% RSLogix 500 project BANCTEST.RSS, saved by version 9.00.00.04 %
PROJECT "BANCTEST"    % processor: SLC 500, 1747-L542 %

PROGRAM FILES
  LAD 2   50 rungs
  LAD 3   16 rungs
  LAD 4   37 rungs
  LAD 5   18 rungs
  LAD 6   36 rungs
  LAD 7   20 rungs
  LAD 8   20 rungs
  LAD 9   15 rungs
  LAD 10   7 rungs
  LAD 11   8 rungs
  LAD 12   10 rungs
  LAD 13   11 rungs
  LAD 14   19 rungs
  LAD 15   13 rungs
  LAD 21   53 rungs
  LAD 22   64 rungs
  LAD 23   50 rungs
  LAD 24   47 rungs
  LAD 16, 17, 18, 19, 20, 25, 26, 27, 28, 29, 30: only END

DATA FILES
  O0 OUTPUT  44 elements
  I1 INPUT  34 elements
  S2 STATUS  164 elements
  B3 BINARY  11 elements
  T4 TIMER  200 elements
  C5 COUNTER  1 elements
  R6 CONTROL  1 elements
  N7 INTEGER  151 elements
  F8 FLOAT  51 elements
  ST20   11 elements
  N21   100 elements
  N22   100 elements
  N23   51 elements
  N31   51 elements
  N32   51 elements
  N33   51 elements
  N34   51 elements
  N35   51 elements
  N36   51 elements
  N37   51 elements
  N38   51 elements
  N39   1 elements
  N40   11 elements
  N41   11 elements
  N50   50 elements
  N51   21 elements

LADDER 2
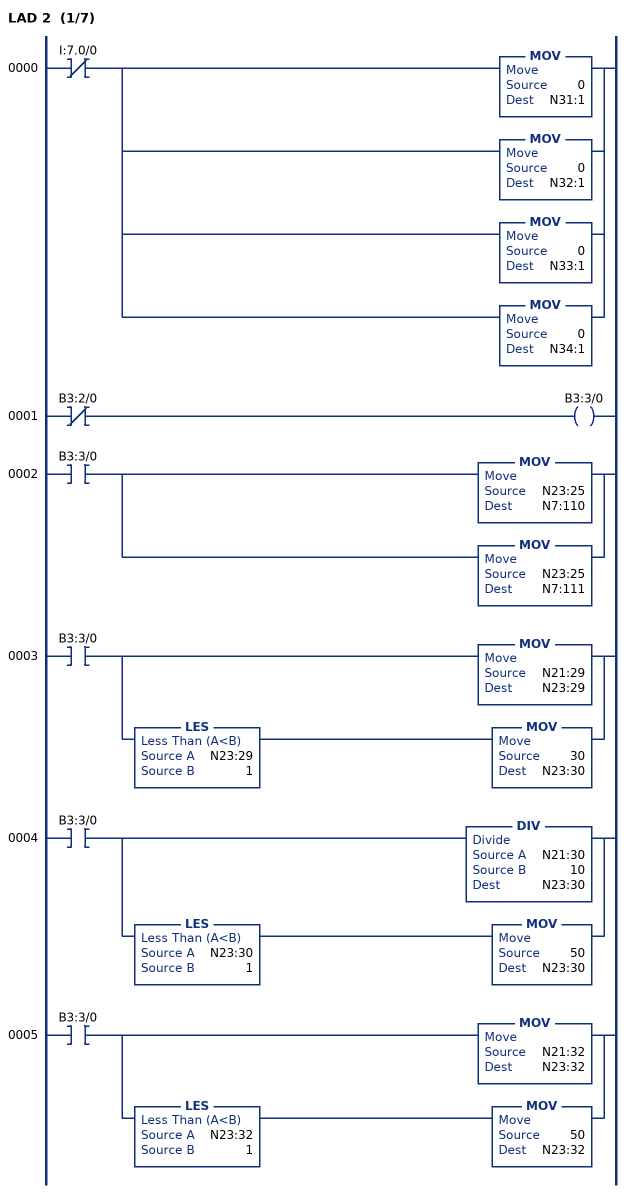
% Rung: 0 %
SOR XIO I:7.0/0 BST MOV 0 N31:1 NXB MOV 0 N32:1 NXB MOV 0 N33:1 NXB MOV 0 N34:1 BND EOR
% Rung: 1 %
SOR XIO B3:2/0 OTE B3:3/0 EOR
% Rung: 2 %
SOR XIC B3:3/0 BST MOV N23:25 N7:110 NXB MOV N23:25 N7:111 BND EOR
% Rung: 3 %
SOR XIC B3:3/0 BST MOV N21:29 N23:29 NXB LES N23:29 1 MOV 30 N23:30 BND EOR
% Rung: 4 %
SOR XIC B3:3/0 BST DIV N21:30 10 N23:30 NXB LES N23:30 1 MOV 50 N23:30 BND EOR
% Rung: 5 %
SOR XIC B3:3/0 BST MOV N21:32 N23:32 NXB LES N23:32 1 MOV 50 N23:32 BND EOR

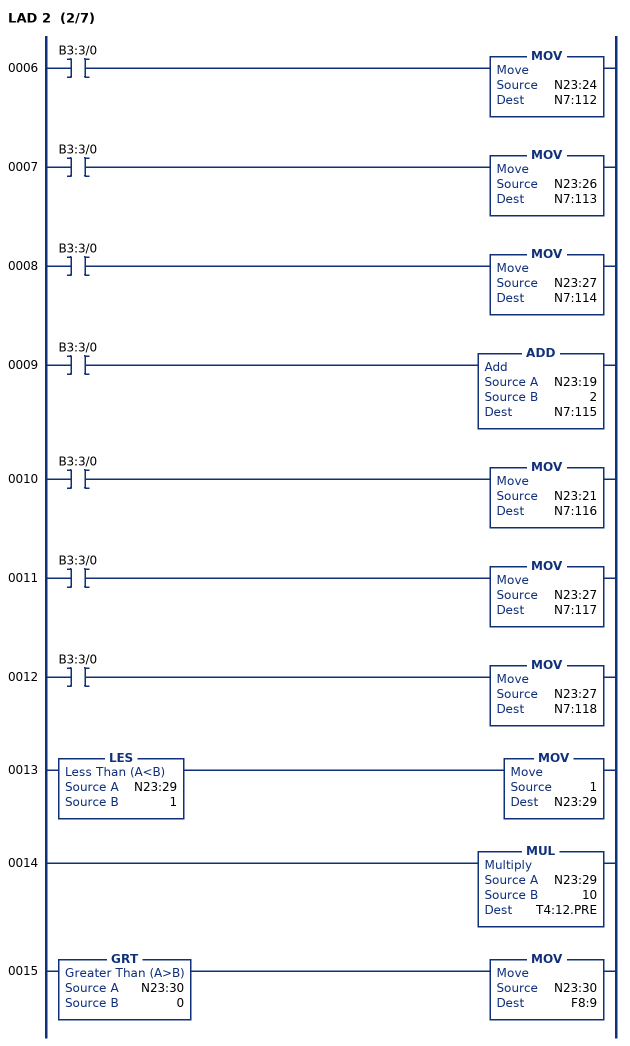
% Rung: 6 %
SOR XIC B3:3/0 MOV N23:24 N7:112 EOR
% Rung: 7 %
SOR XIC B3:3/0 MOV N23:26 N7:113 EOR
% Rung: 8 %
SOR XIC B3:3/0 MOV N23:27 N7:114 EOR
% Rung: 9 %
SOR XIC B3:3/0 ADD N23:19 2 N7:115 EOR
% Rung: 10 %
SOR XIC B3:3/0 MOV N23:21 N7:116 EOR
% Rung: 11 %
SOR XIC B3:3/0 MOV N23:27 N7:117 EOR
% Rung: 12 %
SOR XIC B3:3/0 MOV N23:27 N7:118 EOR
% Rung: 13 %
SOR LES N23:29 1 MOV 1 N23:29 EOR
% Rung: 14 %
SOR MUL N23:29 10 T4:12.PRE EOR
% Rung: 15 %
SOR GRT N23:30 0 MOV N23:30 F8:9 EOR

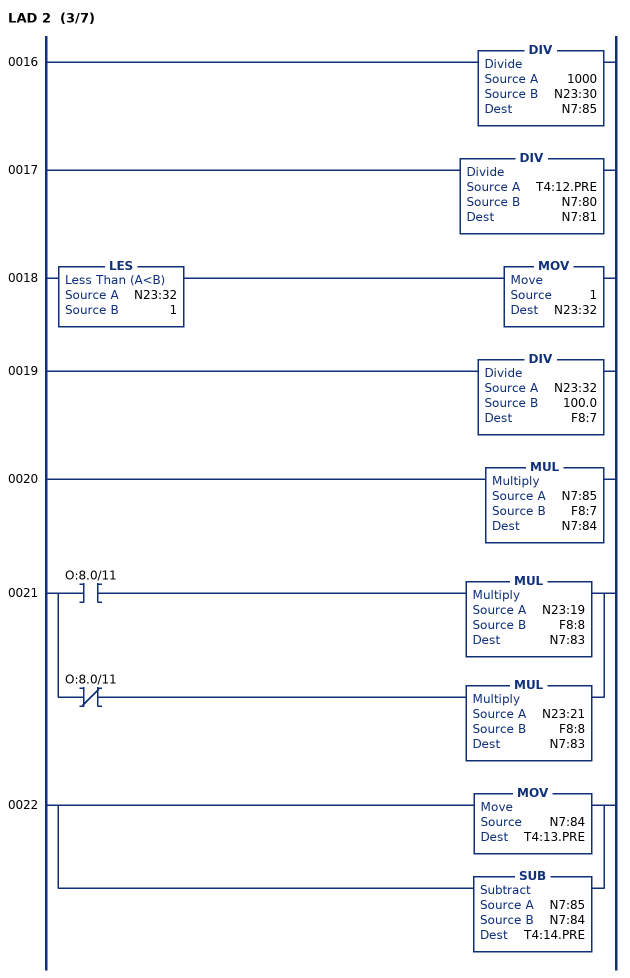
% Rung: 16 %
SOR DIV 1000 N23:30 N7:85 EOR
% Rung: 17 %
SOR DIV T4:12.PRE N7:80 N7:81 EOR
% Rung: 18 %
SOR LES N23:32 1 MOV 1 N23:32 EOR
% Rung: 19 %
SOR DIV N23:32 100.0 F8:7 EOR
% Rung: 20 %
SOR MUL N7:85 F8:7 N7:84 EOR
% Rung: 21 %
SOR BST XIC O:8.0/11 MUL N23:19 F8:8 N7:83 NXB XIO O:8.0/11 MUL N23:21 F8:8 N7:83 BND EOR
% Rung: 22 %
SOR BST MOV N7:84 T4:13.PRE NXB SUB N7:85 N7:84 T4:14.PRE BND EOR

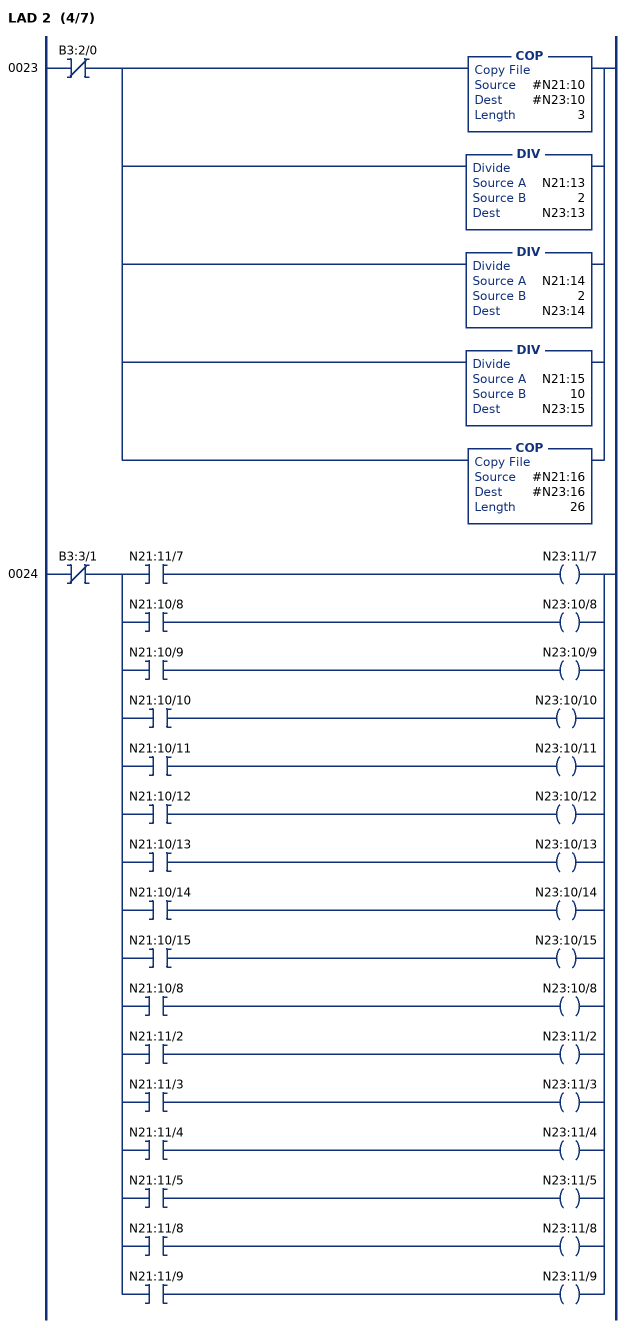
% Rung: 23 %
SOR XIO B3:2/0 BST COP #N21:10 #N23:10 3 NXB DIV N21:13 2 N23:13 NXB DIV N21:14 2 N23:14 NXB DIV N21:15 10 N23:15 NXB COP #N21:16 #N23:16 26 BND EOR
% Rung: 24 %
SOR XIO B3:3/1 BST XIC N21:11/7 OTE N23:11/7 NXB XIC N21:10/8 OTE N23:10/8 NXB XIC N21:10/9 OTE N23:10/9 NXB XIC N21:10/10 OTE N23:10/10 NXB XIC N21:10/11 OTE N23:10/11 NXB XIC N21:10/12 OTE N23:10/12 NXB XIC N21:10/13 OTE N23:10/13 NXB XIC N21:10/14 OTE N23:10/14 NXB XIC N21:10/15 OTE N23:10/15 NXB XIC N21:10/8 OTE N23:10/8 NXB XIC N21:11/2 OTE N23:11/2 NXB XIC N21:11/3 OTE N23:11/3 NXB XIC N21:11/4 OTE N23:11/4 NXB XIC N21:11/5 OTE N23:11/5 NXB XIC N21:11/8 OTE N23:11/8 NXB XIC N21:11/9 OTE N23:11/9 BND EOR

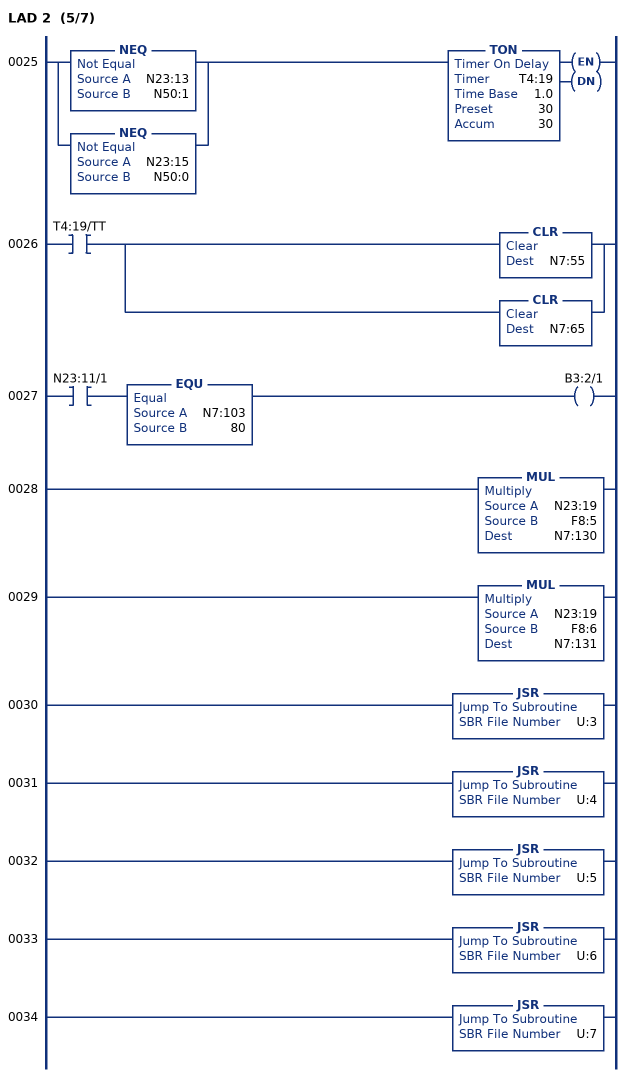
% Rung: 25 %
SOR BST NEQ N23:13 N50:1 NXB NEQ N23:15 N50:0 BND TON T4:19 1.0 30 30 EOR
% Rung: 26 %
SOR XIC T4:19/TT BST CLR N7:55 NXB CLR N7:65 BND EOR
% Rung: 27 %
SOR XIC N23:11/1 EQU N7:103 80 OTE B3:2/1 EOR
% Rung: 28 %
SOR MUL N23:19 F8:5 N7:130 EOR
% Rung: 29 %
SOR MUL N23:19 F8:6 N7:131 EOR
% Rung: 30 %
SOR JSR U:3 EOR
% Rung: 31 %
SOR JSR U:4 EOR
% Rung: 32 %
SOR JSR U:5 EOR
% Rung: 33 %
SOR JSR U:6 EOR
% Rung: 34 %
SOR JSR U:7 EOR

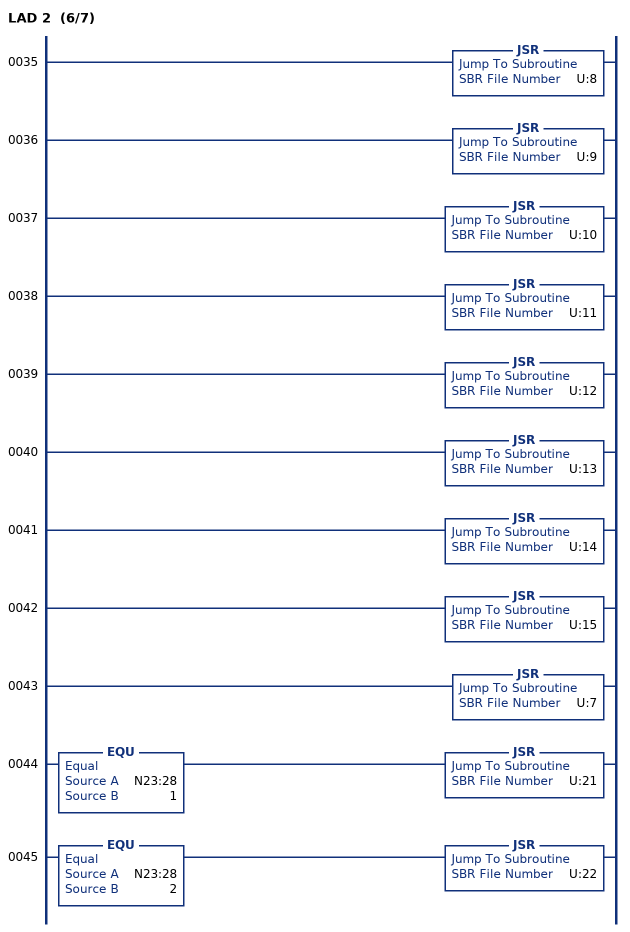
% Rung: 35 %
SOR JSR U:8 EOR
% Rung: 36 %
SOR JSR U:9 EOR
% Rung: 37 %
SOR JSR U:10 EOR
% Rung: 38 %
SOR JSR U:11 EOR
% Rung: 39 %
SOR JSR U:12 EOR
% Rung: 40 %
SOR JSR U:13 EOR
% Rung: 41 %
SOR JSR U:14 EOR
% Rung: 42 %
SOR JSR U:15 EOR
% Rung: 43 %
SOR JSR U:7 EOR
% Rung: 44 %
SOR EQU N23:28 1 JSR U:21 EOR
% Rung: 45 %
SOR EQU N23:28 2 JSR U:22 EOR

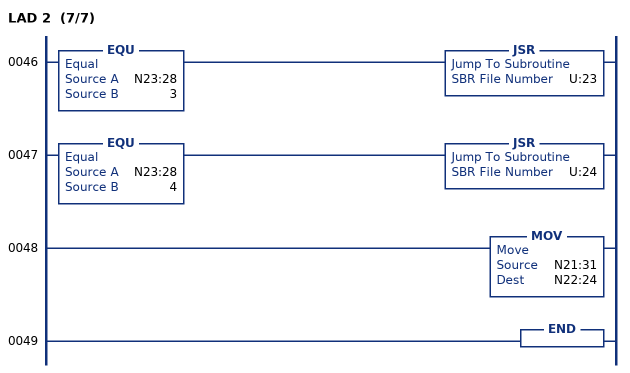
% Rung: 46 %
SOR EQU N23:28 3 JSR U:23 EOR
% Rung: 47 %
SOR EQU N23:28 4 JSR U:24 EOR
% Rung: 48 %
SOR MOV N21:31 N22:24 EOR
% Rung: 49 %
SOR END EOR

LADDER 3
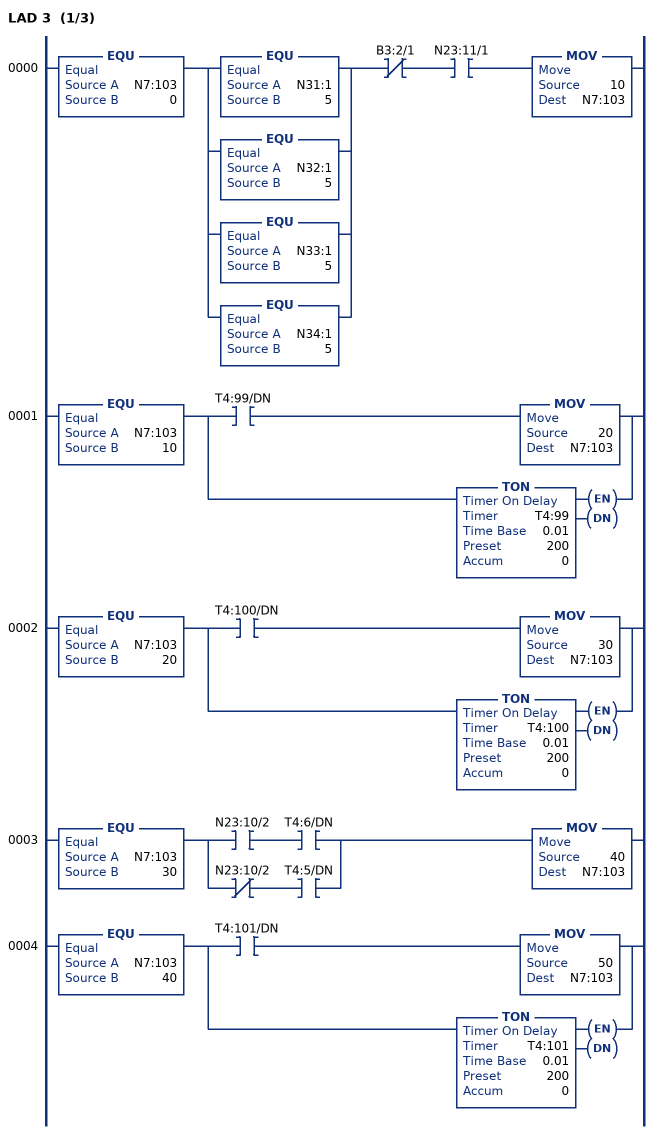
% Rung: 0 %
SOR EQU N7:103 0 BST EQU N31:1 5 NXB EQU N32:1 5 NXB EQU N33:1 5 NXB EQU N34:1 5 BND XIO B3:2/1 XIC N23:11/1 MOV 10 N7:103 EOR
% Rung: 1 %
SOR EQU N7:103 10 BST XIC T4:99/DN MOV 20 N7:103 NXB TON T4:99 0.01 200 0 BND EOR
% Rung: 2 %
SOR EQU N7:103 20 BST XIC T4:100/DN MOV 30 N7:103 NXB TON T4:100 0.01 200 0 BND EOR
% Rung: 3 %
SOR EQU N7:103 30 BST XIC N23:10/2 XIC T4:6/DN NXB XIO N23:10/2 XIC T4:5/DN BND MOV 40 N7:103 EOR
% Rung: 4 %
SOR EQU N7:103 40 BST XIC T4:101/DN MOV 50 N7:103 NXB TON T4:101 0.01 200 0 BND EOR

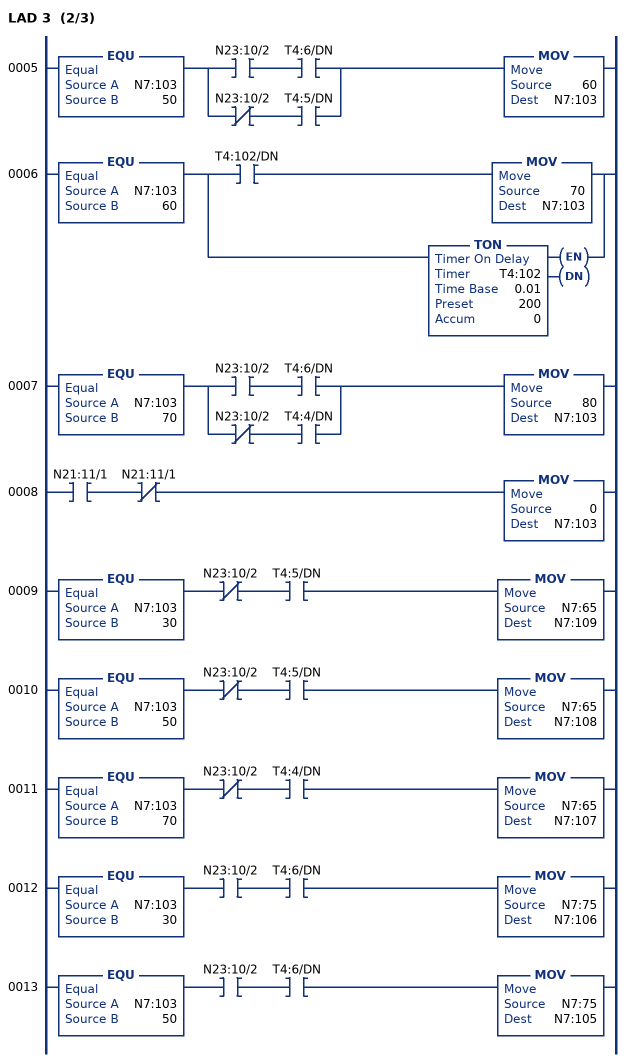
% Rung: 5 %
SOR EQU N7:103 50 BST XIC N23:10/2 XIC T4:6/DN NXB XIO N23:10/2 XIC T4:5/DN BND MOV 60 N7:103 EOR
% Rung: 6 %
SOR EQU N7:103 60 BST XIC T4:102/DN MOV 70 N7:103 NXB TON T4:102 0.01 200 0 BND EOR
% Rung: 7 %
SOR EQU N7:103 70 BST XIC N23:10/2 XIC T4:6/DN NXB XIO N23:10/2 XIC T4:4/DN BND MOV 80 N7:103 EOR
% Rung: 8 %
SOR XIC N21:11/1 XIO N21:11/1 MOV 0 N7:103 EOR
% Rung: 9 %
SOR EQU N7:103 30 XIO N23:10/2 XIC T4:5/DN MOV N7:65 N7:109 EOR
% Rung: 10 %
SOR EQU N7:103 50 XIO N23:10/2 XIC T4:5/DN MOV N7:65 N7:108 EOR
% Rung: 11 %
SOR EQU N7:103 70 XIO N23:10/2 XIC T4:4/DN MOV N7:65 N7:107 EOR
% Rung: 12 %
SOR EQU N7:103 30 XIC N23:10/2 XIC T4:6/DN MOV N7:75 N7:106 EOR
% Rung: 13 %
SOR EQU N7:103 50 XIC N23:10/2 XIC T4:6/DN MOV N7:75 N7:105 EOR

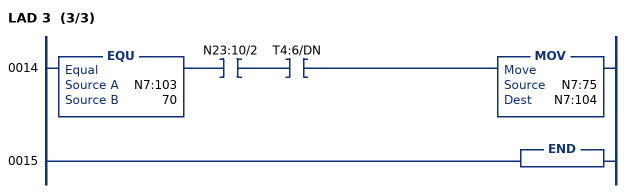
% Rung: 14 %
SOR EQU N7:103 70 XIC N23:10/2 XIC T4:6/DN MOV N7:75 N7:104 EOR
% Rung: 15 %
SOR END EOR

LADDER 4
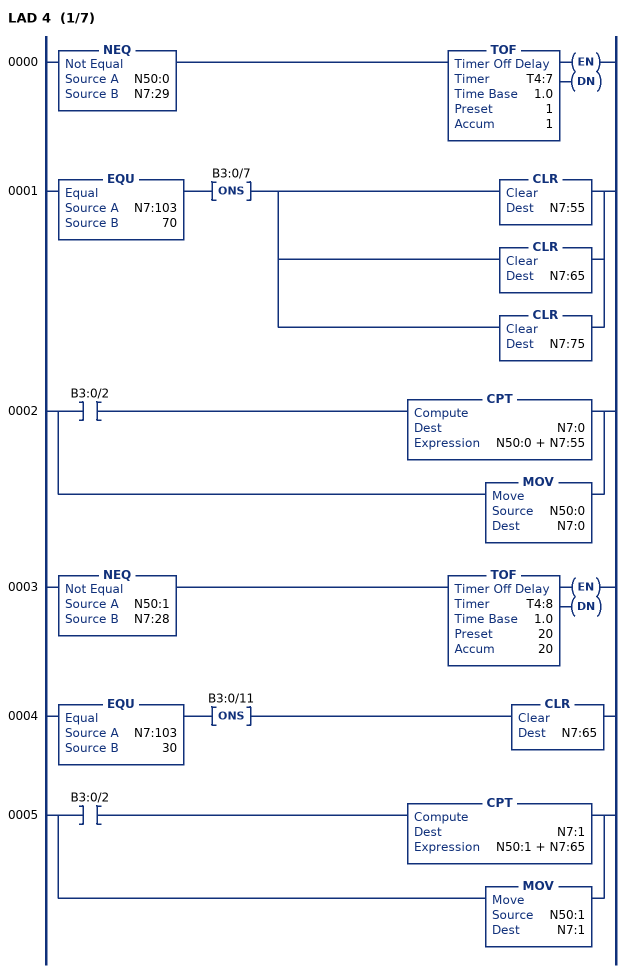
% Rung: 0 %
SOR NEQ N50:0 N7:29 TOF T4:7 1.0 1 1 EOR
% Rung: 1 %
SOR EQU N7:103 70 OSR B3:0/7 BST CLR N7:55 NXB CLR N7:65 NXB CLR N7:75 BND EOR
% Rung: 2 %
SOR BST XIC B3:0/2 CPT N7:0 " N50:0 + N7:55 " NXB MOV N50:0 N7:0 BND EOR
% Rung: 3 %
SOR NEQ N50:1 N7:28 TOF T4:8 1.0 20 20 EOR
% Rung: 4 %
SOR EQU N7:103 30 OSR B3:0/11 CLR N7:65 EOR
% Rung: 5 %
SOR BST XIC B3:0/2 CPT N7:1 " N50:1 + N7:65 " NXB MOV N50:1 N7:1 BND EOR

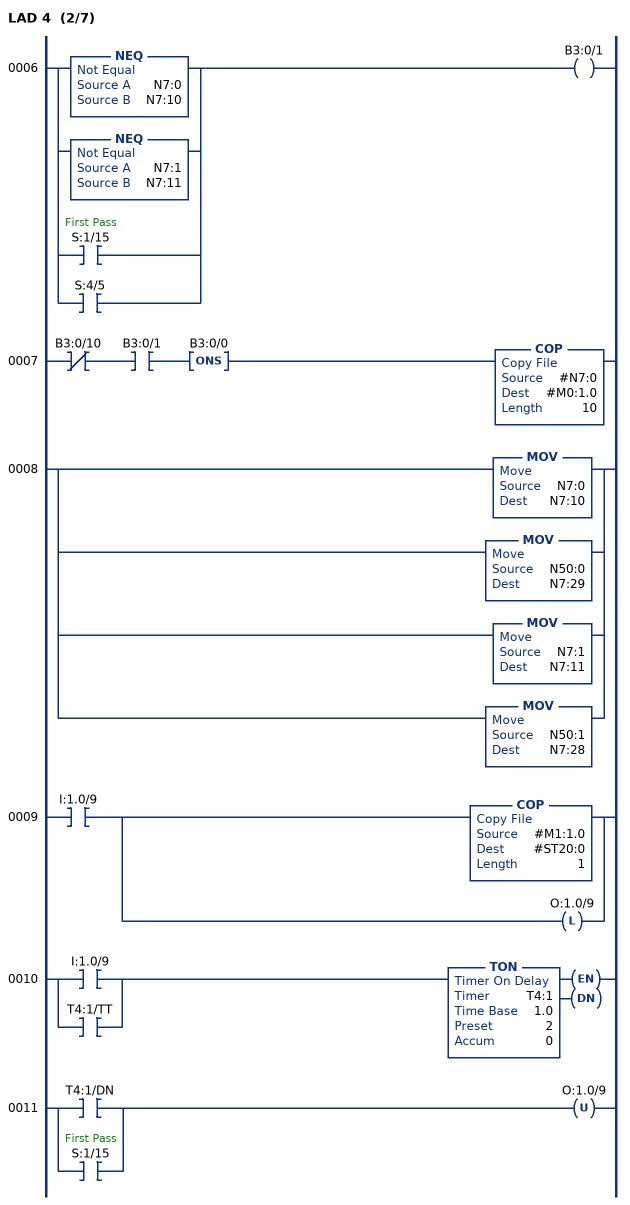
% Rung: 6 %
SOR BST NEQ N7:0 N7:10 NXB NEQ N7:1 N7:11 NXB XIC S:1/15 NXB XIC S:4/5 BND OTE B3:0/1 EOR
%   S:1/15  "First Pass" %
% Rung: 7 %
SOR XIO B3:0/10 XIC B3:0/1 OSR B3:0/0 COP #N7:0 #M0:1.0 10 EOR
% Rung: 8 %
SOR BST MOV N7:0 N7:10 NXB MOV N50:0 N7:29 NXB MOV N7:1 N7:11 NXB MOV N50:1 N7:28 BND EOR
% Rung: 9 %
SOR XIC I:1.0/9 BST COP #M1:1.0 #ST20:0 1 NXB OTL O:1.0/9 BND EOR
% Rung: 10 %
SOR BST XIC I:1.0/9 NXB XIC T4:1/TT BND TON T4:1 1.0 2 0 EOR
% Rung: 11 %
SOR BST XIC T4:1/DN NXB XIC S:1/15 BND OTU O:1.0/9 EOR
%   S:1/15  "First Pass" %

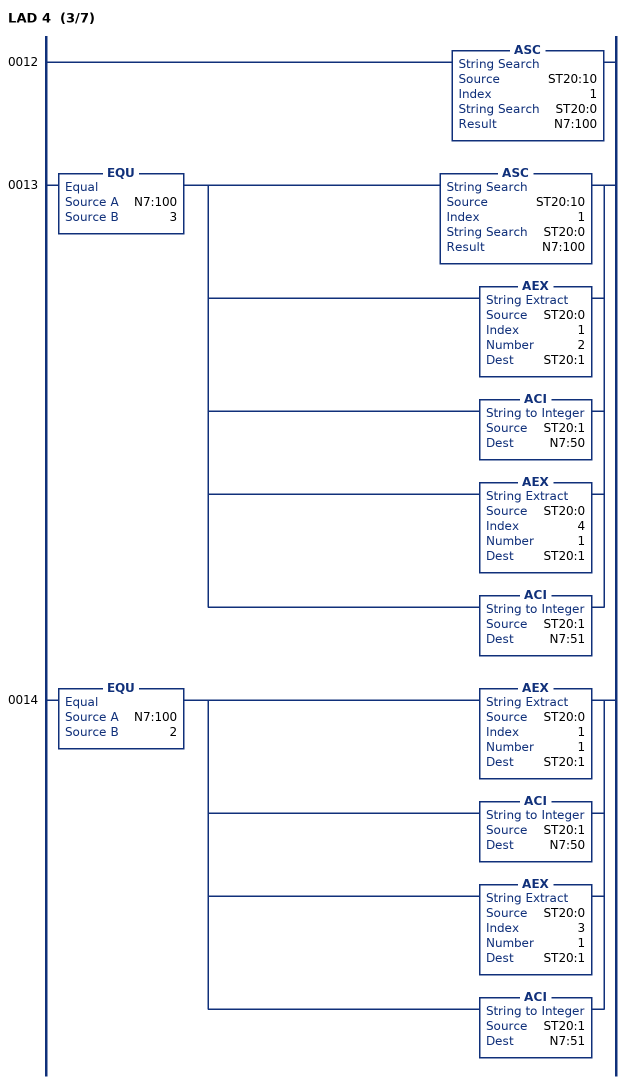
% Rung: 12 %
SOR ASC ST20:10 1 ST20:0 N7:100 EOR
% Rung: 13 %
SOR EQU N7:100 3 BST ASC ST20:10 1 ST20:0 N7:100 NXB AEX ST20:0 1 2 ST20:1 NXB ACI ST20:1 N7:50 NXB AEX ST20:0 4 1 ST20:1 NXB ACI ST20:1 N7:51 BND EOR
% Rung: 14 %
SOR EQU N7:100 2 BST AEX ST20:0 1 1 ST20:1 NXB ACI ST20:1 N7:50 NXB AEX ST20:0 3 1 ST20:1 NXB ACI ST20:1 N7:51 BND EOR

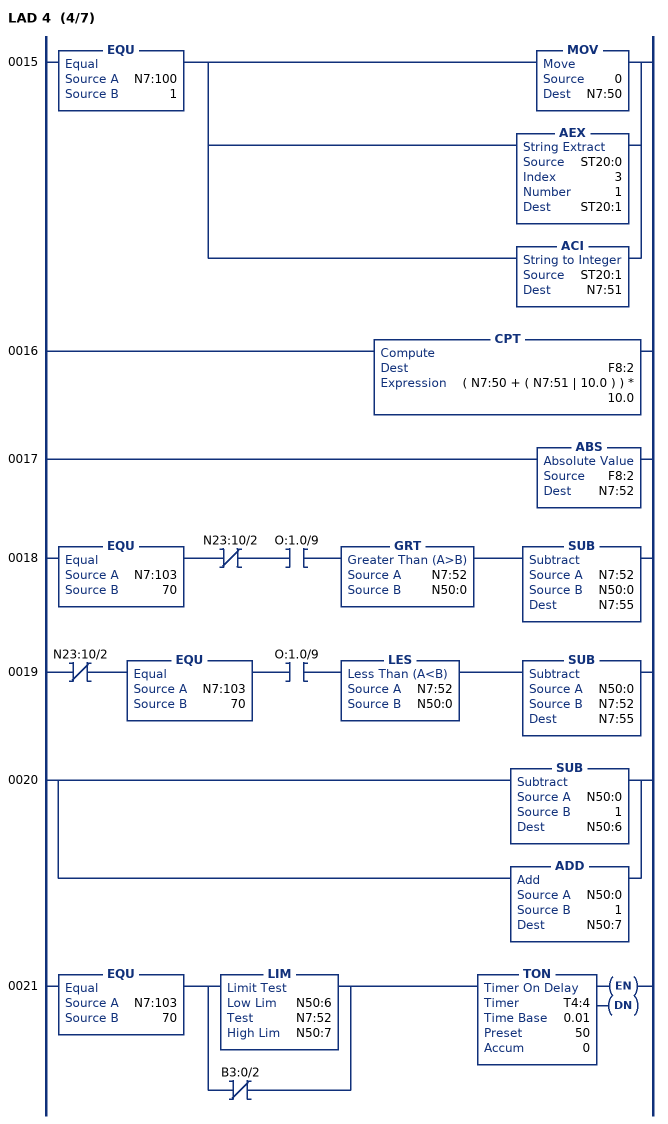
% Rung: 15 %
SOR EQU N7:100 1 BST MOV 0 N7:50 NXB AEX ST20:0 3 1 ST20:1 NXB ACI ST20:1 N7:51 BND EOR
% Rung: 16 %
SOR CPT F8:2 " ( N7:50 + ( N7:51 | 10.0 ) ) * 10.0 " EOR
% Rung: 17 %
SOR ABS F8:2 N7:52 EOR
% Rung: 18 %
SOR EQU N7:103 70 XIO N23:10/2 XIC O:1.0/9 GRT N7:52 N50:0 SUB N7:52 N50:0 N7:55 EOR
% Rung: 19 %
SOR XIO N23:10/2 EQU N7:103 70 XIC O:1.0/9 LES N7:52 N50:0 SUB N50:0 N7:52 N7:55 EOR
% Rung: 20 %
SOR BST SUB N50:0 1 N50:6 NXB ADD N50:0 1 N50:7 BND EOR
% Rung: 21 %
SOR EQU N7:103 70 BST LIM N50:6 N7:52 N50:7 NXB XIO B3:0/2 BND TON T4:4 0.01 50 0 EOR

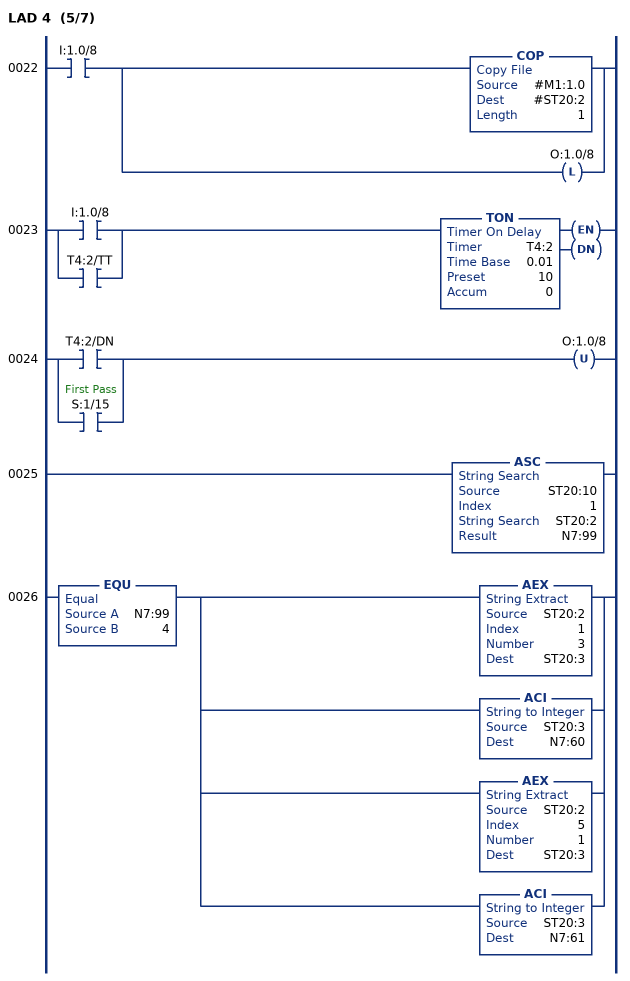
% Rung: 22 %
SOR XIC I:1.0/8 BST COP #M1:1.0 #ST20:2 1 NXB OTL O:1.0/8 BND EOR
% Rung: 23 %
SOR BST XIC I:1.0/8 NXB XIC T4:2/TT BND TON T4:2 0.01 10 0 EOR
% Rung: 24 %
SOR BST XIC T4:2/DN NXB XIC S:1/15 BND OTU O:1.0/8 EOR
%   S:1/15  "First Pass" %
% Rung: 25 %
SOR ASC ST20:10 1 ST20:2 N7:99 EOR
% Rung: 26 %
SOR EQU N7:99 4 BST AEX ST20:2 1 3 ST20:3 NXB ACI ST20:3 N7:60 NXB AEX ST20:2 5 1 ST20:3 NXB ACI ST20:3 N7:61 BND EOR

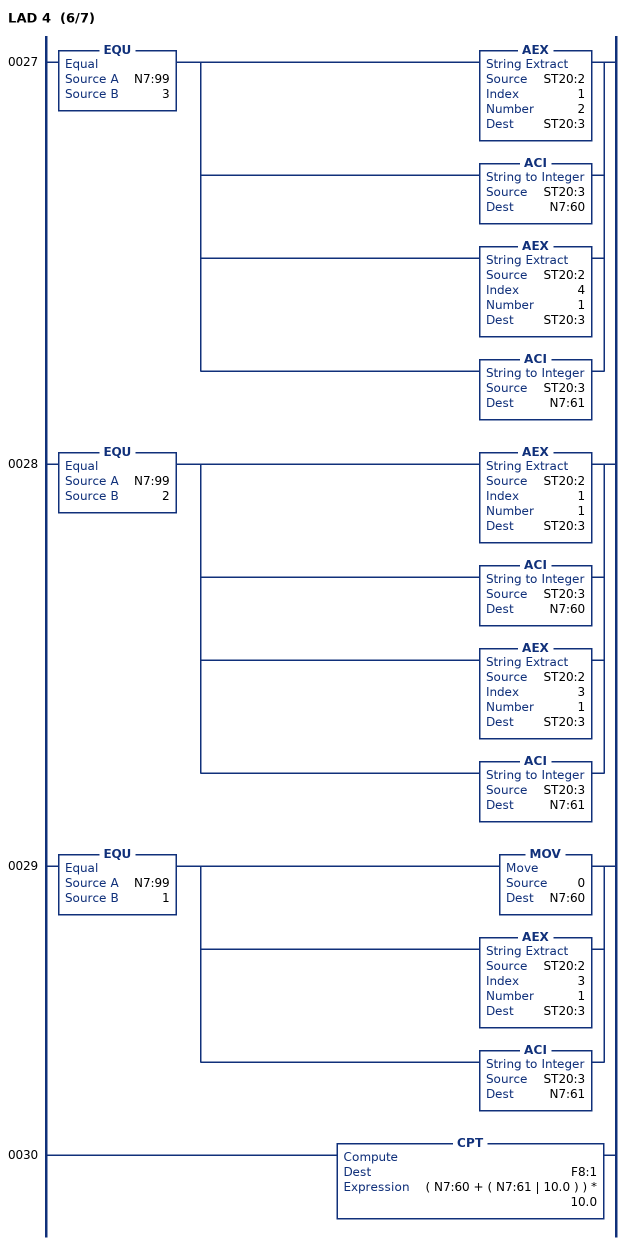
% Rung: 27 %
SOR EQU N7:99 3 BST AEX ST20:2 1 2 ST20:3 NXB ACI ST20:3 N7:60 NXB AEX ST20:2 4 1 ST20:3 NXB ACI ST20:3 N7:61 BND EOR
% Rung: 28 %
SOR EQU N7:99 2 BST AEX ST20:2 1 1 ST20:3 NXB ACI ST20:3 N7:60 NXB AEX ST20:2 3 1 ST20:3 NXB ACI ST20:3 N7:61 BND EOR
% Rung: 29 %
SOR EQU N7:99 1 BST MOV 0 N7:60 NXB AEX ST20:2 3 1 ST20:3 NXB ACI ST20:3 N7:61 BND EOR
% Rung: 30 %
SOR CPT F8:1 " ( N7:60 + ( N7:61 | 10.0 ) ) * 10.0 " EOR

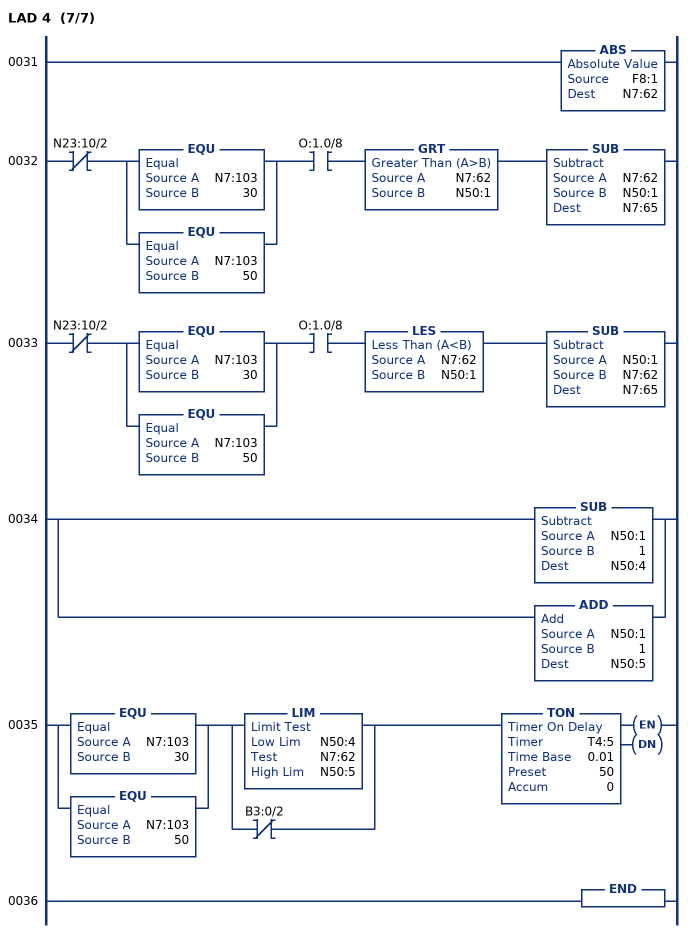
% Rung: 31 %
SOR ABS F8:1 N7:62 EOR
% Rung: 32 %
SOR XIO N23:10/2 BST EQU N7:103 30 NXB EQU N7:103 50 BND XIC O:1.0/8 GRT N7:62 N50:1 SUB N7:62 N50:1 N7:65 EOR
% Rung: 33 %
SOR XIO N23:10/2 BST EQU N7:103 30 NXB EQU N7:103 50 BND XIC O:1.0/8 LES N7:62 N50:1 SUB N50:1 N7:62 N7:65 EOR
% Rung: 34 %
SOR BST SUB N50:1 1 N50:4 NXB ADD N50:1 1 N50:5 BND EOR
% Rung: 35 %
SOR BST EQU N7:103 30 NXB EQU N7:103 50 BND BST LIM N50:4 N7:62 N50:5 NXB XIO B3:0/2 BND TON T4:5 0.01 50 0 EOR
% Rung: 36 %
SOR END EOR

LADDER 5
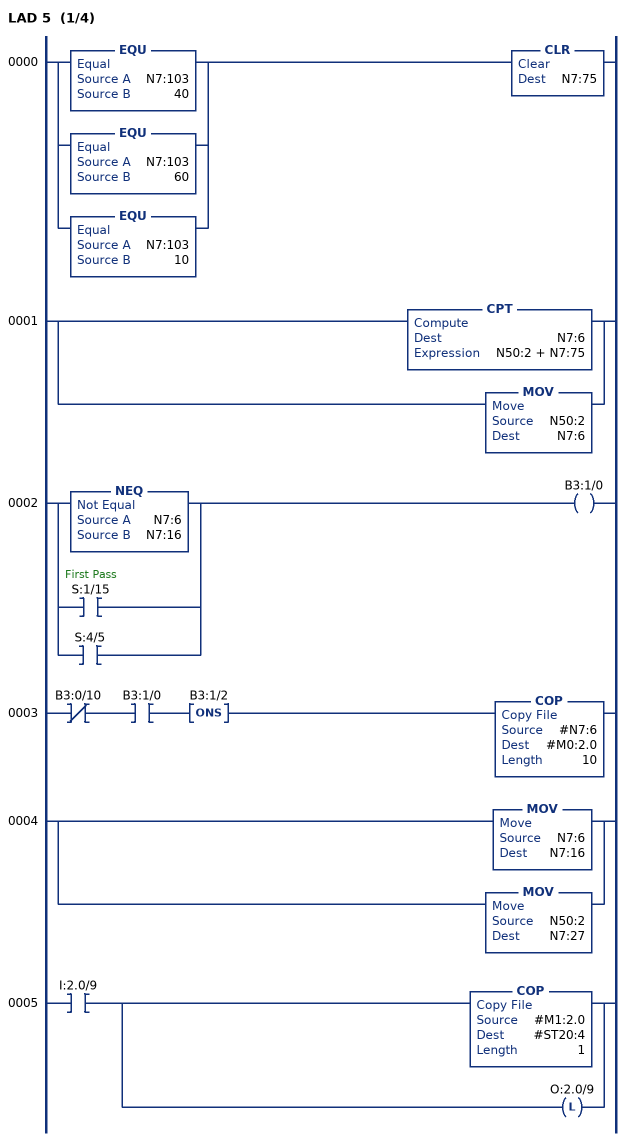
% Rung: 0 %
SOR BST EQU N7:103 40 NXB EQU N7:103 60 NXB EQU N7:103 10 BND CLR N7:75 EOR
% Rung: 1 %
SOR BST CPT N7:6 " N50:2 + N7:75 " NXB MOV N50:2 N7:6 BND EOR
% Rung: 2 %
SOR BST NEQ N7:6 N7:16 NXB XIC S:1/15 NXB XIC S:4/5 BND OTE B3:1/0 EOR
%   S:1/15  "First Pass" %
% Rung: 3 %
SOR XIO B3:0/10 XIC B3:1/0 OSR B3:1/2 COP #N7:6 #M0:2.0 10 EOR
% Rung: 4 %
SOR BST MOV N7:6 N7:16 NXB MOV N50:2 N7:27 BND EOR
% Rung: 5 %
SOR XIC I:2.0/9 BST COP #M1:2.0 #ST20:4 1 NXB OTL O:2.0/9 BND EOR

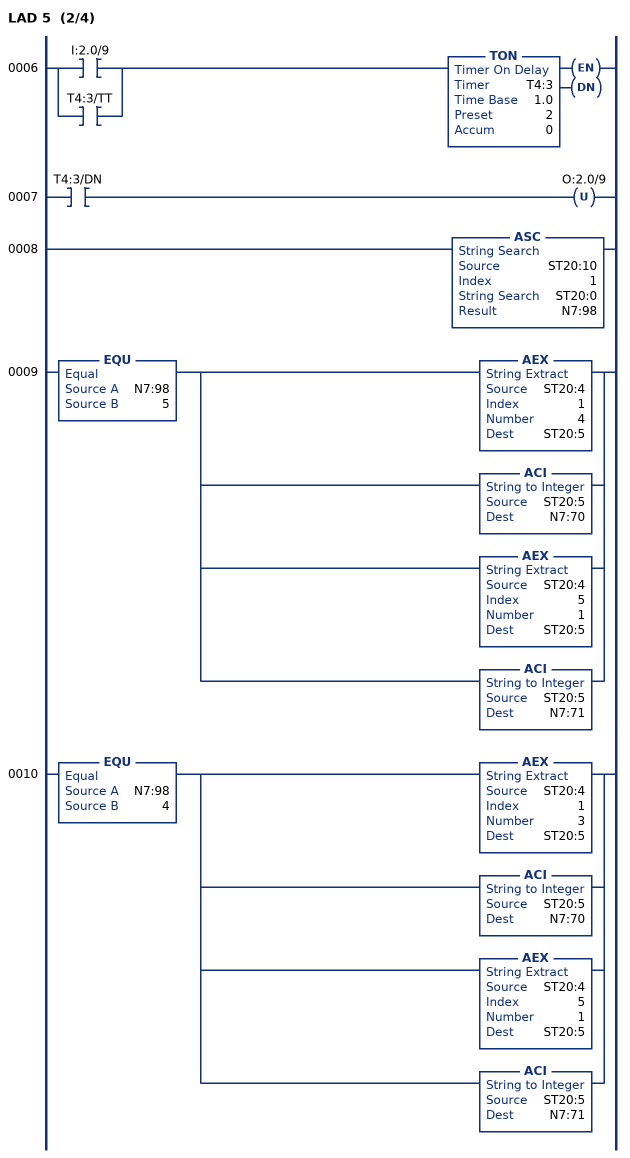
% Rung: 6 %
SOR BST XIC I:2.0/9 NXB XIC T4:3/TT BND TON T4:3 1.0 2 0 EOR
% Rung: 7 %
SOR XIC T4:3/DN OTU O:2.0/9 EOR
% Rung: 8 %
SOR ASC ST20:10 1 ST20:0 N7:98 EOR
% Rung: 9 %
SOR EQU N7:98 5 BST AEX ST20:4 1 4 ST20:5 NXB ACI ST20:5 N7:70 NXB AEX ST20:4 5 1 ST20:5 NXB ACI ST20:5 N7:71 BND EOR
% Rung: 10 %
SOR EQU N7:98 4 BST AEX ST20:4 1 3 ST20:5 NXB ACI ST20:5 N7:70 NXB AEX ST20:4 5 1 ST20:5 NXB ACI ST20:5 N7:71 BND EOR

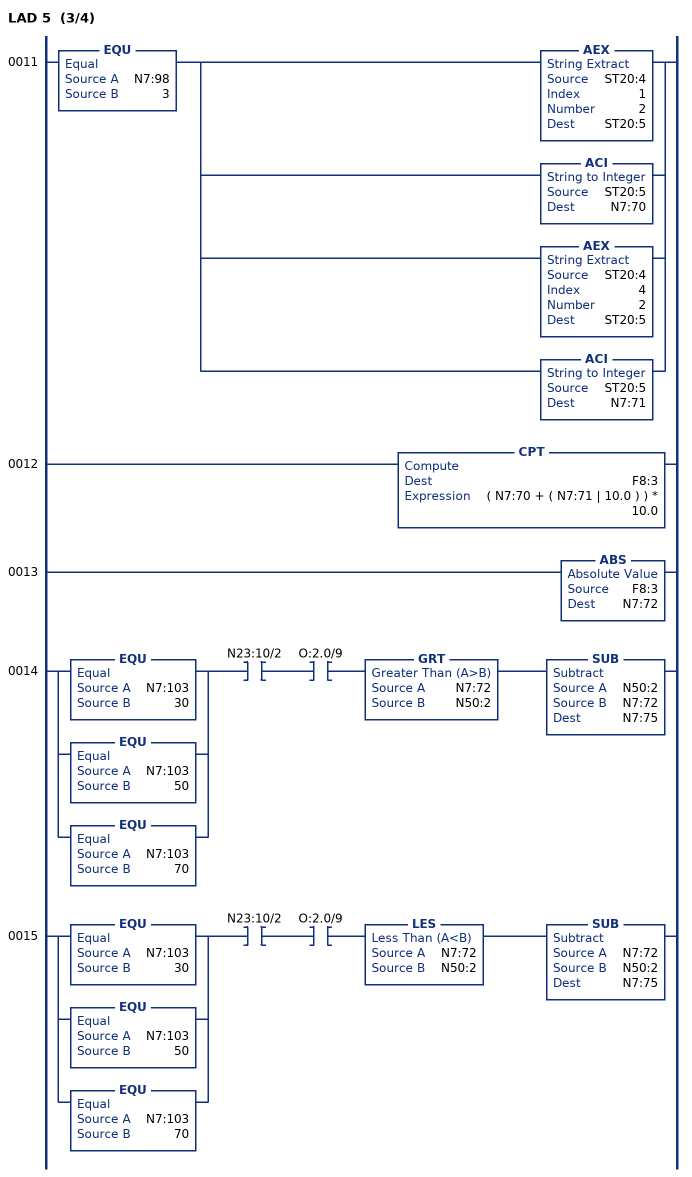
% Rung: 11 %
SOR EQU N7:98 3 BST AEX ST20:4 1 2 ST20:5 NXB ACI ST20:5 N7:70 NXB AEX ST20:4 4 2 ST20:5 NXB ACI ST20:5 N7:71 BND EOR
% Rung: 12 %
SOR CPT F8:3 " ( N7:70 + ( N7:71 | 10.0 ) ) * 10.0 " EOR
% Rung: 13 %
SOR ABS F8:3 N7:72 EOR
% Rung: 14 %
SOR BST EQU N7:103 30 NXB EQU N7:103 50 NXB EQU N7:103 70 BND XIC N23:10/2 XIC O:2.0/9 GRT N7:72 N50:2 SUB N50:2 N7:72 N7:75 EOR
% Rung: 15 %
SOR BST EQU N7:103 30 NXB EQU N7:103 50 NXB EQU N7:103 70 BND XIC N23:10/2 XIC O:2.0/9 LES N7:72 N50:2 SUB N7:72 N50:2 N7:75 EOR

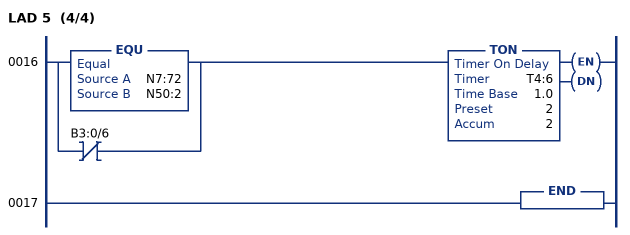
% Rung: 16 %
SOR BST EQU N7:72 N50:2 NXB XIO B3:0/6 BND TON T4:6 1.0 2 2 EOR
% Rung: 17 %
SOR END EOR

LADDER 6
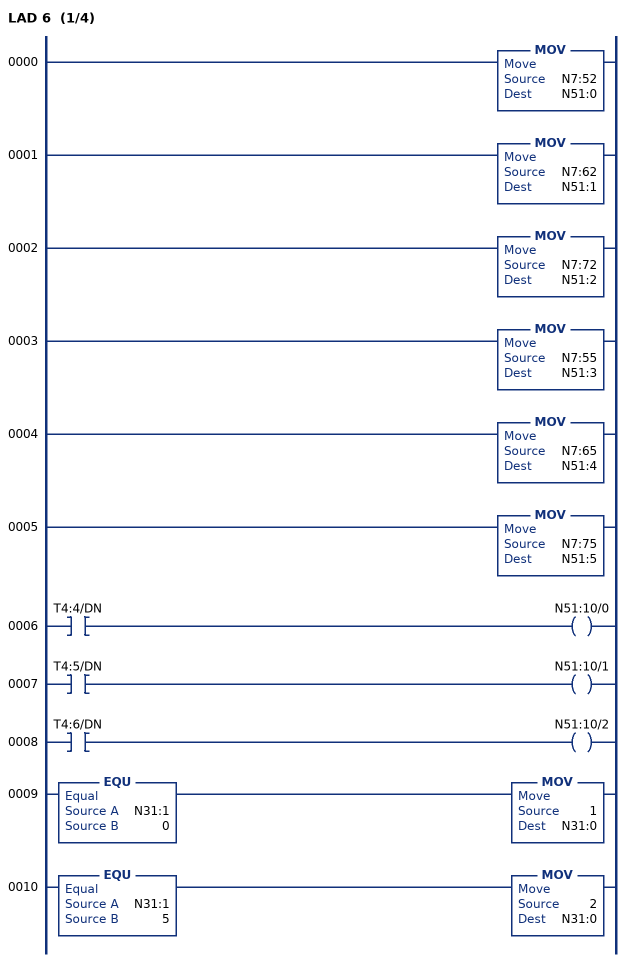
% Rung: 0 %
SOR MOV N7:52 N51:0 EOR
% Rung: 1 %
SOR MOV N7:62 N51:1 EOR
% Rung: 2 %
SOR MOV N7:72 N51:2 EOR
% Rung: 3 %
SOR MOV N7:55 N51:3 EOR
% Rung: 4 %
SOR MOV N7:65 N51:4 EOR
% Rung: 5 %
SOR MOV N7:75 N51:5 EOR
% Rung: 6 %
SOR XIC T4:4/DN OTE N51:10/0 EOR
% Rung: 7 %
SOR XIC T4:5/DN OTE N51:10/1 EOR
% Rung: 8 %
SOR XIC T4:6/DN OTE N51:10/2 EOR
% Rung: 9 %
SOR EQU N31:1 0 MOV 1 N31:0 EOR
% Rung: 10 %
SOR EQU N31:1 5 MOV 2 N31:0 EOR

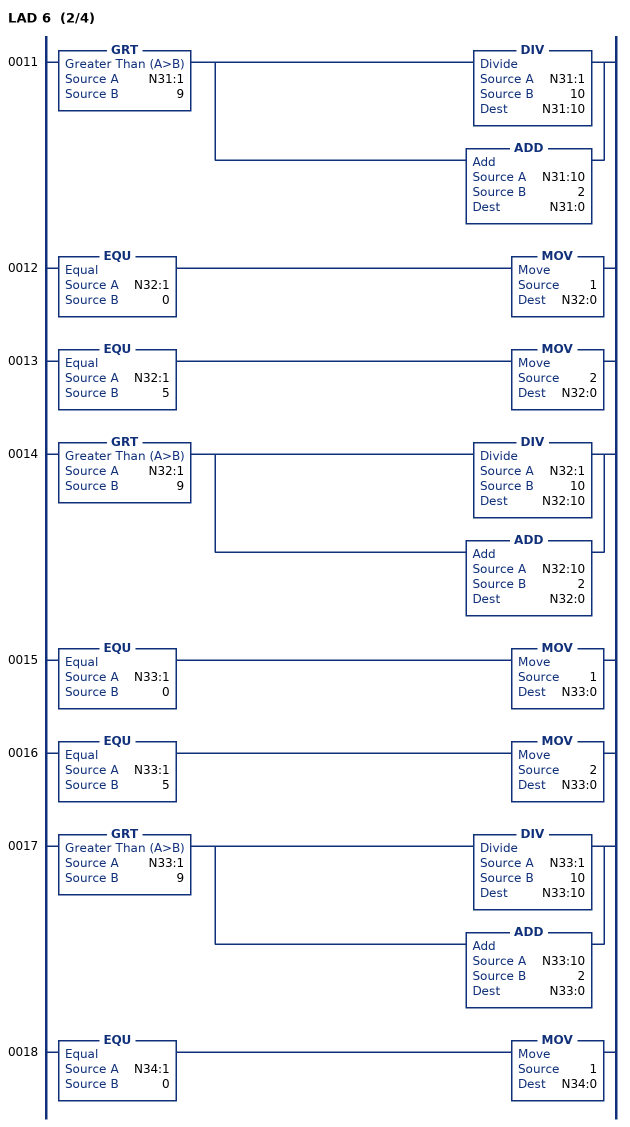
% Rung: 11 %
SOR GRT N31:1 9 BST DIV N31:1 10 N31:10 NXB ADD N31:10 2 N31:0 BND EOR
% Rung: 12 %
SOR EQU N32:1 0 MOV 1 N32:0 EOR
% Rung: 13 %
SOR EQU N32:1 5 MOV 2 N32:0 EOR
% Rung: 14 %
SOR GRT N32:1 9 BST DIV N32:1 10 N32:10 NXB ADD N32:10 2 N32:0 BND EOR
% Rung: 15 %
SOR EQU N33:1 0 MOV 1 N33:0 EOR
% Rung: 16 %
SOR EQU N33:1 5 MOV 2 N33:0 EOR
% Rung: 17 %
SOR GRT N33:1 9 BST DIV N33:1 10 N33:10 NXB ADD N33:10 2 N33:0 BND EOR
% Rung: 18 %
SOR EQU N34:1 0 MOV 1 N34:0 EOR

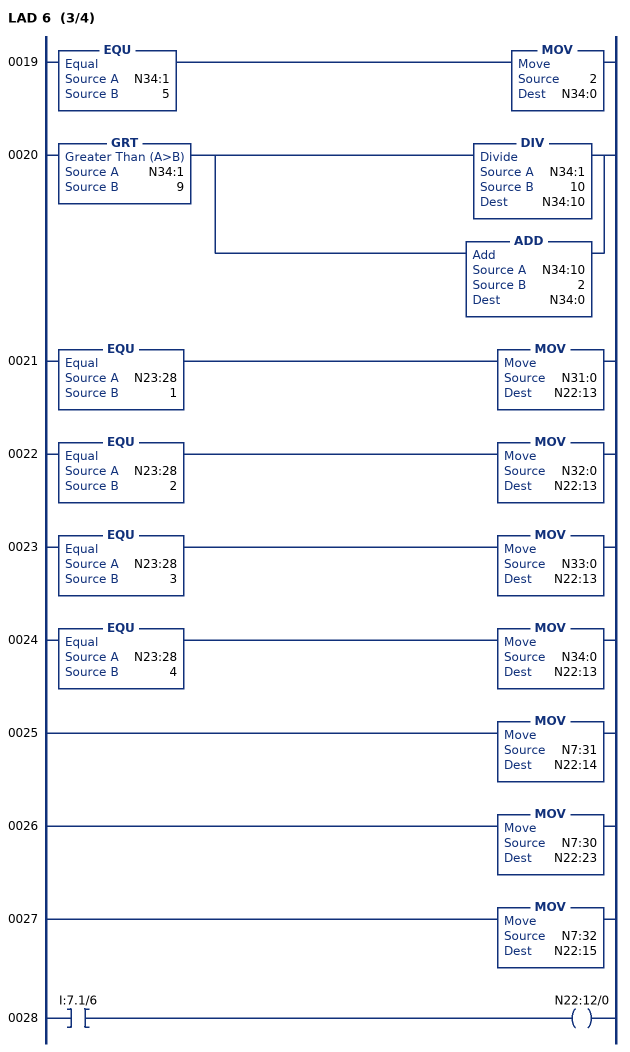
% Rung: 19 %
SOR EQU N34:1 5 MOV 2 N34:0 EOR
% Rung: 20 %
SOR GRT N34:1 9 BST DIV N34:1 10 N34:10 NXB ADD N34:10 2 N34:0 BND EOR
% Rung: 21 %
SOR EQU N23:28 1 MOV N31:0 N22:13 EOR
% Rung: 22 %
SOR EQU N23:28 2 MOV N32:0 N22:13 EOR
% Rung: 23 %
SOR EQU N23:28 3 MOV N33:0 N22:13 EOR
% Rung: 24 %
SOR EQU N23:28 4 MOV N34:0 N22:13 EOR
% Rung: 25 %
SOR MOV N7:31 N22:14 EOR
% Rung: 26 %
SOR MOV N7:30 N22:23 EOR
% Rung: 27 %
SOR MOV N7:32 N22:15 EOR
% Rung: 28 %
SOR XIC I:7.1/6 OTE N22:12/0 EOR

